Staubli VAL3: cmdDisableOp.pgx

public program cmdDisableOp(num x_nAxNum)
begin
  //发送“终止操作”指令到所选驱动器
  if bOpeEnabled[x_nAxNum]==true
    doFaultReset[x_nAxNum]=false
    doEnableOp[x_nAxNum]=false
    delay(0.1)
    doQuickStop[x_nAxNum]=true
    doEnableVoltage[x_nAxNum]=true
    doSwitchOn[x_nAxNum]=true
  endIf
end
